INTERFACE PUBLIC Writer EXTENDS __SYSTEM.IQueryInterface

END_INTERFACE

(* stored: Version 1.1.0.1
   Itf Writer: Id {718875e1-2b42-48f4-a770-215689a441f4} *)
